FUNCTION_BLOCK FB_AnalogLoadCellInput
VAR_INPUT
	rYIntercept : REAL := -72.1; // Y intercept when fitting a line for Integer Counts (Y) v.s. Applied Mass (X) 
	rXSlope : REAL := -371; // Slope when fitting a line for Integer Coutns (Y) v.s. Applied Mass (X)
	sUnits : STRING := 'N'; 
END_VAR
VAR_OUTPUT
	nRawCounts : INT; // Copied from nAnalogReading
	rCalibratedOutput : REAL; 
	sOutputUnits : STRING; // Copied from sUnits 
END_VAR
VAR
	nAnalogReading AT %I* : INT; 
END_VAR

// First get the analog reading, and save it 
nRawCounts := nAnalogReading; 

// Then, convert the reading to get the output in calibrated format: 
rCalibratedOutput := (nRawCounts - rYIntercept) * (1/(rXSlope)); 

// Finally, copy over the units 
sOutputUnits := sUnits;

END_FUNCTION_BLOCK

(* stored: Version 1.1.0.1, ProductVersion 3.1.4024.12
   POU FB_AnalogLoadCellInput: Id {4a41d613-ff1c-4eac-a4f4-deb57692fb09}, SpecialFunc None *)
